TYPE ST_HES_Parameter :
STRUCT
	Temp_Kuehlwasser_Max		: REAL;
	Temp_Kuehlwasser_Min		: REAL;

	AutoQuittierung				: BOOL;
	Sollwert					: REAL;
END_STRUCT
END_TYPE

(* stored: Version 1.1.0.1, ProductVersion 3.1.4024.9
   DUT ST_HES_Parameter: Id {da31c80e-7263-4acb-95e9-2b5eb21cb271} *)
